{attribute 'GeneratedUsingTerminal: EL1512-0000-0017'}
{attribute addProperty BoxType "EL1512-0000-0017"}
{attribute addProperty Id "EtcSlaveTerminalBaseCNT_Inputs_Channel_1AT %I*CNT_Inputs_Channel_54FF2F1E8CNT_Inputs_Channel_2AT %I*CNT_Inputs_Channel_54FF2F1E8CNT_Outputs_Channel_1AT %Q*CNT_Outputs_Channel_550BB6DF6CNT_Outputs_Channel_2AT %Q*CNT_Outputs_Channel_550BB6DF6WcStateAT %I*WcState_9091E0EB2InfoDataAT %I*InfoData_32EB74EA10"}
{attribute addProperty CRC "790734071"}
{attribute addProperty Size "40"}
TYPE EL1512_2F21A4F7 EXTENDS EtcSlaveTerminalBase :
STRUCT
	{attribute addProperty Name "CNT_Inputs_Channel_1"}
	CNT_Inputs_Channel_1 : CNT_Inputs_Channel_54FF2F1E;
	{attribute addProperty Name "CNT_Inputs_Channel_2"}
	CNT_Inputs_Channel_2 : CNT_Inputs_Channel_54FF2F1E;
	{attribute addProperty Name "CNT_Outputs_Channel_1"}
	CNT_Outputs_Channel_1 : CNT_Outputs_Channel_550BB6DF;
	{attribute addProperty Name "CNT_Outputs_Channel_2"}
	CNT_Outputs_Channel_2 : CNT_Outputs_Channel_550BB6DF;
	{attribute addProperty Name "WcState"}
	WcState : WcState_9091E0EB;
	{attribute addProperty Name "InfoData"}
	InfoData : InfoData_32EB74EA;
END_STRUCT
END_TYPE

(* stored: Version 1.2.0.0, ProductVersion 3.1.4024.9
   DUT EL1512_2F21A4F7: Id {ffd2e38d-c26c-4cea-a82c-28bd75234554} *)
